(* IEC 61131-3 sources: beckhoffAutomationInterface/ST/Shark/Lib/BehaviorTree/decorators, 6 files *)

(* ---- FB_ForceFailureNode.st ---- *)
FUNCTION_BLOCK FB_ForceFailureNode IMPLEMENTS I_TreeNode
VAR
    _ipChild : I_TreeNode;
END_VAR

METHOD PUBLIC SetChild : BOOL
VAR_INPUT
    ipChild : I_TreeNode;
END_VAR
    _ipChild := ipChild;
    SetChild := TRUE;
END_METHOD

METHOD Tick : ST_NodeResult
VAR
    stChildStatus : ST_NodeResult;
END_VAR
    IF _ipChild <> 0 THEN
        stChildStatus := _ipChild.Tick();
        IF stChildStatus.eStatus = E_NodeStatus.RUNNING THEN
            Tick := stChildStatus;
        ELSE
            // ForceFailure doesn't propagate child error - it's intentional failure
            Tick.eStatus := E_NodeStatus.FAILURE;
            Tick.sDescription := CONCAT('Forced Failure after: ', stChildStatus.sDescription);
            Tick.rProgress := stChildStatus.rProgress;
        END_IF
    ELSE
        Tick.eStatus := E_NodeStatus.FAILURE;
        Tick.sDescription := 'ForceFailure missing child';
    END_IF
END_METHOD

{attribute 'estimated-stack-usage' := '500'}
METHOD Halt
    IF _ipChild <> 0 THEN
        _ipChild.Halt();
    END_IF
END_METHOD

{attribute 'estimated-stack-usage' := '500'}
METHOD Reset : BOOL
    IF _ipChild <> 0 THEN
        _ipChild.Reset();
    END_IF
    Reset := TRUE;
END_METHOD

END_FUNCTION_BLOCK

(* ---- FB_ForceSuccessNode.st ---- *)
FUNCTION_BLOCK FB_ForceSuccessNode IMPLEMENTS I_TreeNode
VAR
    _ipChild : I_TreeNode;
END_VAR

METHOD PUBLIC SetChild : BOOL
VAR_INPUT
    ipChild : I_TreeNode;
END_VAR
    _ipChild := ipChild;
    SetChild := TRUE;
END_METHOD

METHOD Tick : ST_NodeResult
VAR
    stChildStatus : ST_NodeResult;
END_VAR
    IF _ipChild <> 0 THEN
        stChildStatus := _ipChild.Tick();
        IF stChildStatus.eStatus = E_NodeStatus.RUNNING THEN
            Tick := stChildStatus;
        ELSE
            Tick.eStatus := E_NodeStatus.SUCCESS;
            Tick.sDescription := CONCAT('Forced Success after: ', stChildStatus.sDescription);
            Tick.rProgress := 100.0;
        END_IF
    ELSE
        Tick.eStatus := E_NodeStatus.SUCCESS;
        Tick.sDescription := 'ForceSuccess missing child';
        Tick.rProgress := 100.0;
    END_IF
END_METHOD

{attribute 'estimated-stack-usage' := '500'}
METHOD Halt
    IF _ipChild <> 0 THEN
        _ipChild.Halt();
    END_IF
END_METHOD

{attribute 'estimated-stack-usage' := '500'}
METHOD Reset : BOOL
    IF _ipChild <> 0 THEN
        _ipChild.Reset();
    END_IF
    Reset := TRUE;
END_METHOD

END_FUNCTION_BLOCK

(* ---- FB_InverterNode.st ---- *)
FUNCTION_BLOCK FB_InverterNode IMPLEMENTS I_TreeNode
VAR_INPUT
    sName : STRING(50) := 'Inverter';
END_VAR
VAR
    _ipChild : I_TreeNode;
END_VAR

METHOD PUBLIC SetChild : BOOL
VAR_INPUT
    ipNode : I_TreeNode;
END_VAR
    IF ipNode = 0 THEN
        SetChild := FALSE;
        RETURN;
    END_IF
    _ipChild := ipNode;
    SetChild := TRUE;
END_METHOD

METHOD Tick : ST_NodeResult
VAR
    stChildStatus : ST_NodeResult;
END_VAR
    IF _ipChild = 0 THEN
        Tick := F_BuildNullChildResult(sName, 'Inverter child not configured');
        RETURN;
    END_IF

    stChildStatus := _ipChild.Tick();
    Tick := stChildStatus; // copies error and progress naturally

    // Inverter swaps SUCCESS<->FAILURE
    IF stChildStatus.eStatus = E_NodeStatus.SUCCESS THEN
        Tick.eStatus := E_NodeStatus.FAILURE;
        Tick.sDescription := CONCAT('Inverted SUCCESS: ', stChildStatus.sDescription);
    ELSIF stChildStatus.eStatus = E_NodeStatus.FAILURE THEN
        Tick.eStatus := E_NodeStatus.SUCCESS;
        Tick.bHasError := FALSE; // clear error!
        Tick.stError.eErrorId := E_ErrorId.NO_ERROR;
        Tick.sDescription := CONCAT('Inverted FAILURE: ', stChildStatus.sDescription);
    END_IF
END_METHOD

{attribute 'estimated-stack-usage' := '500'}
METHOD Halt
    IF _ipChild <> 0 THEN
        _ipChild.Halt();
    END_IF
END_METHOD

{attribute 'estimated-stack-usage' := '500'}
METHOD Reset : BOOL
    IF _ipChild <> 0 THEN
        Reset := _ipChild.Reset();
    ELSE
        Reset := TRUE;
    END_IF
END_METHOD

END_FUNCTION_BLOCK

(* ---- FB_RepeatNode.st ---- *)
FUNCTION_BLOCK FB_RepeatNode IMPLEMENTS I_TreeNode
VAR_INPUT
    sName : STRING(50) := 'Repeat Node';
    nNumCycles : INT := 3; // -1 for infinite
END_VAR
VAR
    _ipChild : I_TreeNode;
    _nCycles : INT := 0;
END_VAR

METHOD PUBLIC SetChild : BOOL
VAR_INPUT
    ipChild : I_TreeNode;
END_VAR
    _ipChild := ipChild;
    SetChild := TRUE;
END_METHOD

    {attribute 'estimated-stack-usage' := '500'}
METHOD Tick : ST_NodeResult
VAR
    stChildStatus : ST_NodeResult;
END_VAR
    IF _ipChild = 0 THEN
        Tick := F_BuildNullChildResult(sName, 'Repeat decorator child not configured');
        RETURN;
    END_IF

    stChildStatus := _ipChild.Tick();

    IF stChildStatus.eStatus = E_NodeStatus.FAILURE THEN
        // Propagate child error
        Tick := stChildStatus;
        IF NOT Tick.bHasError THEN
            Tick.bHasError := TRUE;
            Tick.stError.eErrorId := E_ErrorId.ERR_BT_CHILD_FAILED;
            Tick.stError.sSource := sName;
            Tick.stError.sMessage := 'Repeat child failed';
        END_IF
        _nCycles := 0;
        RETURN;
    ELSIF stChildStatus.eStatus = E_NodeStatus.SUCCESS THEN
        _nCycles := _nCycles + 1;
        IF nNumCycles <> -1 AND _nCycles >= nNumCycles THEN
            _nCycles := 0;
            Tick.eStatus := E_NodeStatus.SUCCESS;
            Tick.rProgress := 100.0;
            Tick.sDescription := CONCAT('Completed ', TO_STRING(nNumCycles));
            Tick.sDescription := CONCAT(Tick.sDescription, ' cycles');
        ELSE
            _ipChild.Reset();
            Tick.eStatus := E_NodeStatus.RUNNING; // Keep repeating
            Tick.sDescription := CONCAT('Repeating sequence: ', TO_STRING(_nCycles));

            // Progress: completed cycles + child sub-progress
            IF nNumCycles > 0 THEN
                Tick.rProgress := (INT_TO_REAL(_nCycles) / INT_TO_REAL(nNumCycles)) * 100.0;
            END_IF
        END_IF
    ELSE
        Tick.eStatus := E_NodeStatus.RUNNING;
        Tick.sDescription := stChildStatus.sDescription;

        // Child still running — blend cycle progress with child sub-progress
        IF nNumCycles > 0 THEN
            Tick.rProgress := (INT_TO_REAL(_nCycles) + stChildStatus.rProgress / 100.0) / INT_TO_REAL(nNumCycles) * 100.0;
        END_IF
    END_IF

END_METHOD

// Method: Halt - Stops execution but preserves error state
{attribute 'estimated-stack-usage' := '500'}
{attribute 'estimated-stack-usage' := '500'}
METHOD Halt
    _nCycles := 0;
    IF _ipChild <> 0 THEN
        _ipChild.Halt();
    END_IF
END_METHOD

    {attribute 'estimated-stack-usage' := '500'}
METHOD Reset : BOOL
    IF _ipChild <> 0 THEN
        _ipChild.Reset();
    END_IF
    Reset := TRUE;
END_METHOD

END_FUNCTION_BLOCK

(* ---- FB_RetryNode.st ---- *)
FUNCTION_BLOCK FB_RetryNode IMPLEMENTS I_TreeNode
VAR_INPUT
    sName : STRING(50) := 'Retry Node';
    nMaxAttempts : INT := 3;
END_VAR
VAR
    _ipChild : I_TreeNode;
    _nAttempts : INT := 0;
END_VAR

METHOD PUBLIC SetChild : BOOL
VAR_INPUT
    ipChild : I_TreeNode;
END_VAR
    _ipChild := ipChild;
    SetChild := TRUE;
END_METHOD

    {attribute 'estimated-stack-usage' := '500'}
METHOD Tick : ST_NodeResult
VAR
    stChildStatus : ST_NodeResult;
    sErrorMsg : STRING(255);
END_VAR
    IF _ipChild = 0 THEN
        Tick := F_BuildNullChildResult(sName, 'Retry decorator child not configured');
        RETURN;
    END_IF

    IF nMaxAttempts <= 0 THEN
        Tick.eStatus := E_NodeStatus.FAILURE;
        Tick.bHasError := TRUE;
        Tick.stError.eErrorId := E_ErrorId.ERR_GEN_INVALID_PARAM;
        Tick.stError.sSource := sName;
        Tick.stError.sMessage := 'Retry max attempts must be greater than zero';
        RETURN;
    END_IF

    stChildStatus := _ipChild.Tick();

    IF stChildStatus.eStatus = E_NodeStatus.SUCCESS THEN
        _nAttempts := 0;
        Tick := stChildStatus;
        RETURN;
    ELSIF stChildStatus.eStatus = E_NodeStatus.FAILURE THEN
        _nAttempts := _nAttempts + 1;
        IF _nAttempts < nMaxAttempts THEN
            _ipChild.Reset();
            Tick.eStatus := E_NodeStatus.RUNNING; // Keep trying
            Tick.sDescription := CONCAT('Retrying: attempt ', TO_STRING(_nAttempts));

            // Progress: attempts used so far
            IF nMaxAttempts > 0 THEN
                Tick.rProgress := (INT_TO_REAL(_nAttempts) / INT_TO_REAL(nMaxAttempts)) * 100.0;
            END_IF
        ELSE
            // Max retries exceeded - propagate child error or set generic
            Tick := stChildStatus;

            sErrorMsg := CONCAT('Failed after ', TO_STRING(nMaxAttempts));
            sErrorMsg := CONCAT(sErrorMsg, ' attempts');

            IF NOT Tick.bHasError THEN
                Tick.bHasError := TRUE;
                Tick.stError.eErrorId := E_ErrorId.ERR_BT_MAX_RETRIES;
                Tick.stError.sSource := sName;
            END_IF
            Tick.stError.sMessage := CONCAT(sErrorMsg, CONCAT(': ', Tick.stError.sMessage));

            _nAttempts := 0;
        END_IF
    ELSE
        // Child still running — blend attempt progress with child sub-progress
        Tick.eStatus := E_NodeStatus.RUNNING;
        Tick.sDescription := stChildStatus.sDescription;

        IF nMaxAttempts > 0 THEN
            Tick.rProgress := (INT_TO_REAL(_nAttempts) + stChildStatus.rProgress / 100.0) / INT_TO_REAL(nMaxAttempts) * 100.0;
        END_IF
    END_IF

END_METHOD

    // Method: Halt - Stops execution but preserves error state
{attribute 'estimated-stack-usage' := '500'}
METHOD Halt
    _nAttempts := 0;
    IF _ipChild <> 0 THEN
        _ipChild.Halt();
    END_IF
END_METHOD

{attribute 'estimated-stack-usage' := '500'}
METHOD Reset : BOOL
    _nAttempts := 0;
    IF _ipChild <> 0 THEN
        _ipChild.Reset();
    END_IF
    Reset := TRUE;
END_METHOD

END_FUNCTION_BLOCK

(* ---- FB_TimeoutNode.st ---- *)
FUNCTION_BLOCK FB_TimeoutNode IMPLEMENTS I_TreeNode
VAR_INPUT
    sName : STRING(50) := 'Timeout Node';
    tTimeout : TIME := T#5S;
END_VAR
VAR
    _ipChild : I_TreeNode;
    _fbTimer : TON;
    _bStarted : BOOL := FALSE;
END_VAR

METHOD PUBLIC SetChild : BOOL
VAR_INPUT
    ipChild : I_TreeNode;
END_VAR
    _ipChild := ipChild;
    SetChild := TRUE;
END_METHOD

    {attribute 'estimated-stack-usage' := '500'}
METHOD Tick : ST_NodeResult
VAR
    stChildStatus : ST_NodeResult;
END_VAR
    IF _ipChild = 0 THEN
        Tick := F_BuildNullChildResult(sName, 'Timeout decorator child not configured');
        RETURN;
    END_IF

    // Call timer unconditionally every scan cycle
    _fbTimer(IN := _bStarted, PT := tTimeout);

    IF NOT _bStarted THEN
        _bStarted := TRUE;
    END_IF

    IF _fbTimer.Q THEN
        _ipChild.Halt(); // Stop child but preserve its error state

        Tick.eStatus := E_NodeStatus.FAILURE;
        Tick.bHasError := TRUE;
        Tick.stError.eErrorId := E_ErrorId.ERR_BT_TIMEOUT;
        Tick.stError.sSource := sName;
        Tick.stError.sMessage := CONCAT('Timeout after ', TIME_TO_STRING(tTimeout));
        RETURN;
    END_IF

    stChildStatus := _ipChild.Tick();

    // Track elapsed time as progress (countdown to timeout)
    IF tTimeout > T#0S THEN
        Tick.rProgress := (TIME_TO_REAL(_fbTimer.ET) / TIME_TO_REAL(tTimeout)) * 100.0;
        IF Tick.rProgress > 100.0 THEN Tick.rProgress := 100.0; END_IF
    END_IF

    // Propagate everything exactly from the child
    IF stChildStatus.eStatus <> E_NodeStatus.RUNNING THEN
        _bStarted := FALSE;
        _fbTimer(IN := FALSE);
    END_IF

    Tick.eStatus := stChildStatus.eStatus;
    Tick.bHasError := stChildStatus.bHasError;
    Tick.stError := stChildStatus.stError;
    Tick.sDescription := stChildStatus.sDescription;

    // Use child progress if not overriding it with timer
    IF tTimeout <= T#0S THEN
        Tick.rProgress := stChildStatus.rProgress;
    END_IF

END_METHOD

    // Method: Halt - Stops execution but preserves error state
    {attribute 'estimated-stack-usage' := '200'}
{attribute 'estimated-stack-usage' := '500'}
METHOD Halt
    _bStarted := FALSE;
    _fbTimer(IN := FALSE);
    IF _ipChild <> 0 THEN
        _ipChild.Halt();
    END_IF
END_METHOD

    {attribute 'estimated-stack-usage' := '200'}
METHOD Reset : BOOL
    _bStarted := FALSE;
    _fbTimer(IN := FALSE);
    IF _ipChild <> 0 THEN
        _ipChild.Reset();
    END_IF
    Reset := TRUE;
END_METHOD

END_FUNCTION_BLOCK
